// TIA Portal V19 export
VAR_GLOBAL   // PLC tag table "conveyor-1"
   "Start Button 1" AT %I0.1 : Bool;
   "Stop Button 1" AT %I0.2 : Bool;
   "Belt Conveyor (4m) 1" AT %Q0.1 : Bool;
END_VAR
